VAR_GLOBAL
  gCounter : DINT := 0;
END_VAR

(* stored: Version 1.0
   GVL GVL_Main: Id {00000000-0000-0000-0000-000000000001} *)
